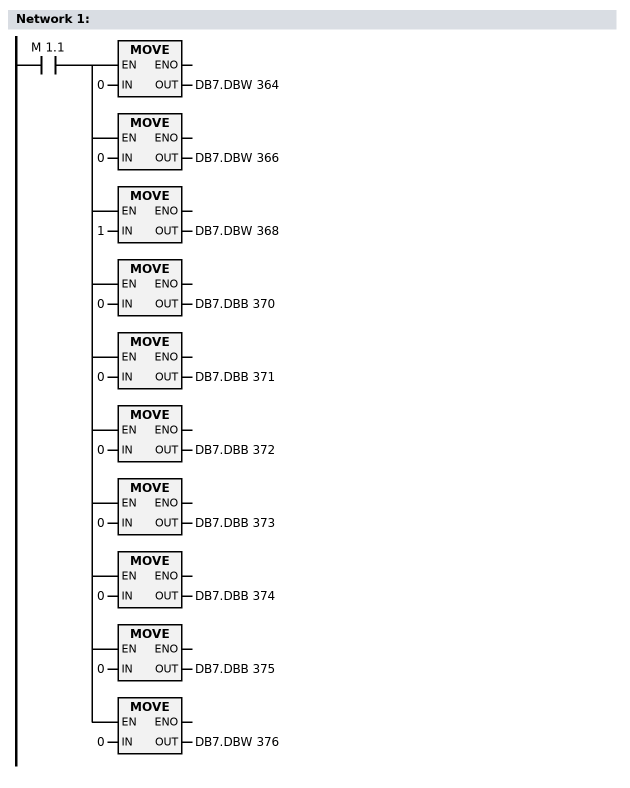
NETWORK
TITLE =
      A     M 1.1;
      =     L 20.0;
      A     L 20.0;
      JNB   M001;
      L     0;
      T     DB7.DBW 364;
M001: NOP   0;
      A     L 20.0;
      JNB   M002;
      L     0;
      T     DB7.DBW 366;
M002: NOP   0;
      A     L 20.0;
      JNB   M003;
      L     1;
      T     DB7.DBW 368;
M003: NOP   0;
      A     L 20.0;
      JNB   M004;
      L     0;
      T     DB7.DBB 370;
M004: NOP   0;
      A     L 20.0;
      JNB   M005;
      L     0;
      T     DB7.DBB 371;
M005: NOP   0;
      A     L 20.0;
      JNB   M006;
      L     0;
      T     DB7.DBB 372;
M006: NOP   0;
      A     L 20.0;
      JNB   M007;
      L     0;
      T     DB7.DBB 373;
M007: NOP   0;
      A     L 20.0;
      JNB   M008;
      L     0;
      T     DB7.DBB 374;
M008: NOP   0;
      A     L 20.0;
      JNB   M009;
      L     0;
      T     DB7.DBB 375;
M009: NOP   0;
      A     L 20.0;
      JNB   M010;
      L     0;
      T     DB7.DBW 376;
M010: NOP   0;
END_ORGANIZATION_BLOCK

ORGANIZATION_BLOCK OB 122
VERSION : 0.1
BEGIN
// (block stored without names or comments; labels and parameter names are numbered)
NETWORK
TITLE =
END_ORGANIZATION_BLOCK
